PROGRAM FB_Blinker
VAR
	fbTimerA: TON;
	fbTimerB: TON;
END_VAR

VAR_INPUT
	bStart: BOOL;
	tSignalTimeOn: TIME;
	tSignalTimeOff: TIME;
END_VAR
VAR_OUTPUT
	bOut: BOOL;
END_VAR

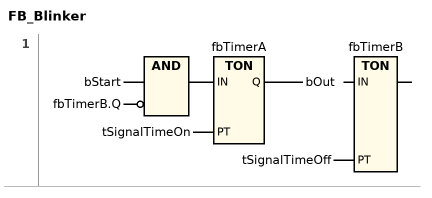
// NETWORK 1
fbTimerA(IN := bStart AND NOT fbTimerB.Q, PT := tSignalTimeOn); // TON
bOut := fbTimerA.Q;
fbTimerB(IN := fbTimerA.Q, PT := tSignalTimeOff); // TON

END_PROGRAM

(* stored: Version 1.1.0.1, ProductVersion 3.1.4024.12
   POU FB_Blinker: Id {eace021f-1441-4f17-8720-39e692f93cf0}, SpecialFunc None *)
